FUNCTION_BLOCK FB_NormallyClosedPB IMPLEMENTS I_Pushbutton
VAR
	Input AT %I* : BOOL;
END_VAR

PROPERTY IsPressed : BOOL
GET
IsPressed := NOT Input;
END_GET
END_PROPERTY

PROPERTY IsReleased : BOOL
GET
IsReleased := Input;
END_GET
END_PROPERTY

END_FUNCTION_BLOCK

(* stored: Version 1.1.0.1, ProductVersion 3.1.4024.9
   POU FB_NormallyClosedPB: Id {03780352-f63e-4023-8055-acbaa9cf7c2e}, SpecialFunc None
   Property IsPressed: Id {03930825-01dd-49c7-98a5-ca54da93f828}
   Get Get: Id {5c983c49-ffab-4ba1-8305-af02090ea6b9}
   Property IsReleased: Id {34dd52bb-0ff9-4c0c-a4a2-01a051380285}
   Get Get: Id {4e3fb3c1-dc7b-4e25-9ad0-968607e778b2} *)
